FUNCTION_BLOCK Station EXTENDS Objective IMPLEMENTS iObjective
VAR	
	
	myPosition			: LREAL;

END_VAR

PROPERTY CurrentMover : REFERENCE TO Mover
GET
VAR
	
	i				: UINT;

END_VAR

// default to unassigned
CurrentMover REF= 0;

// If any tracked mover is located at the Station, return a handle to the Mover
FOR i := 0 TO GVL.NUM_MOVERS-1 DO
	
	IF TrackedMovers[i] <> 0 AND_THEN ABS( MODABS( TrackedMovers[i]^.AxisReference.NcToPlc.ActPos,GVL.TRACK_LENGTH) - Position ) < 1.0 THEN
		CurrentMover	REF= TrackedMovers[i]^;
	END_IF

END_FOR
END_GET
END_PROPERTY

METHOD Cyclic : BOOL
VAR_INPUT
END_VAR
VAR
	i		: USINT;
END_VAR


// If any movers are no longer destined for this station, remove them from the Tracked Movers list
TrackedMoverCount	:= 0;

FOR i := 0 TO GVL.NUM_MOVERS-1 DO
	
	IF TrackedMovers[i] <> 0 AND_THEN TrackedMovers[i]^.CurrentMoveType <> MoverCommandType_enum.MOVETYPE_STATION THEN
		TrackedMovers[i]	:= 0;
	ELSIF TrackedMovers[i] <> 0 AND_THEN TrackedMovers[i]^.Objective <> InstancePath THEN
		TrackedMovers[i]	:= 0;
	END_IF

END_FOR
END_METHOD

PROPERTY MoverInPosition : BOOL
GET
VAR
	
	i				: UINT;
	
END_VAR

// default to false
MoverInPosition		:= FALSE;

// If any tracked mover is located at the Station, set MoverInPos true 
// todo: should maybe add condition for a maximum velocity as well? ie mover ought to be stopped?
FOR i := 0 TO GVL.NUM_MOVERS-1 DO

	IF TrackedMovers[i] <> 0 AND_THEN ABS( MODABS( TrackedMovers[i]^.AxisReference.NcToPlc.ActPos,GVL.TRACK_LENGTH) - Position ) < 1.0 THEN
		MoverInPosition		:= TRUE;
	END_IF

END_FOR;
END_GET
END_PROPERTY

PROPERTY Position : LREAL
GET


	Position	:= myPosition;
END_GET
SET


	myPosition	:= Position;
END_SET
END_PROPERTY

END_FUNCTION_BLOCK

(* stored: Version 1.1.0.1, ProductVersion 3.1.4024.9
   POU Station: Id {5b67f0b3-4286-49f2-9b21-1e637f521584}, SpecialFunc None
   Folder Methods: Id {6b1e6f0c-25c1-483e-90dd-29f6bdd956e2}
   Folder Properties: Id {0e151499-8bc7-4d0d-acff-abc4339273bc}
   Property CurrentMover: Id {b4e35326-78e7-4021-8c91-b7cb4a0e9212}
   Get Get: Id {e0693b4c-fa5c-4b5f-85a0-f0ea84fe50ab}
   Method Cyclic: Id {ae1d7805-bf3f-45a4-9b82-ce6adba37b33}
   Property MoverInPosition: Id {ccc94bfc-d20e-4ea7-8da8-e0df6797280c}
   Get Get: Id {d401d684-2ca2-4bd9-a954-7ea2efdd18c4}
   Property Position: Id {e062e8cc-9f76-4a77-aea3-5a00085987df}
   Get Get: Id {b470ee7d-dbff-409a-8143-88d3140d1c0f}
   Set Set: Id {69d58698-c7cd-48f7-93aa-293011447caf} *)
